// TIA Portal V20 export
DATA_BLOCK "SBK01"   // DB206
// stored: MemoryReserve 100
   VAR
      "X1-0 No EMG stop: Unwinder" : Bool;
      "X2-1 No EMG stop: Reel cut" : Bool;
      "X3-2 No EMG stop: Vision" : Bool;
      "X4-3 No EMG stop: Conveyor" : Bool;
      "X1-4 reserved" : Bool;
      "X2-5 reserved" : Bool;
      "X3-6 reserved" : Bool;
      "X4-7 reserved" : Bool;
      "X5-0 reserved" : Bool;
      "X6-1 reserved" : Bool;
      "X7-2 reserved" : Bool;
   END_VAR
BEGIN
END_DATA_BLOCK
